FUNCTION_BLOCK AngularAxisWidget
VAR_INPUT
END_VAR
VAR_OUTPUT
    positionSymbol : STRING := '°';
    velocitySymbol : STRING := '°/s';
    base : BaseAxisWidget;
END_VAR
VAR_IN_OUT
    baseRef : AngularAxis;
    ref : AngularAxis;
END_VAR
VAR
END_VAR

base(ref := baseRef);

END_FUNCTION_BLOCK

(* stored: Version 1.1.0.1, ProductVersion 3.1.4018.5
   POU AngularAxisWidget: Id {6b7619a5-866d-4e1a-8e7d-3ea20f4dc191}, SpecialFunc None *)
